  MoveL 585 to (127.63, -206.24, -1) mm, rotated rx -180 ry 0 rz 0 deg; joints [14.907, -52.311, 139.809, 14.927, -86.713, -0.372]
  MoveL 586 to (141.54, -192.34, -1) mm, rotated rx -180 ry 0 rz 0 deg; joints [15.844, -52.517, 140.53, 15.857, -87.219, -0.271]
  MoveL 587 to (229.23, -104.7, -1) mm, rotated rx -180 ry 0 rz 0 deg; joints [22.146, -53.586, 144.524, 22.139, -89.999, 0.626]
  MoveC 588 to (229.67, -104.52, -1) mm, rotated rx -180 ry 0 rz 0 deg; joints [22.166, -53.592, 144.549, 22.159, -90.017, 0.633] to (230.12, -104.7, -1) mm, rotated rx -180 ry 0 rz 0 deg; joints [22.165, -53.6, 144.584, 22.159, -90.042, 0.644]
  MoveL 589 to (230.57, -105.15, -1) mm, rotated rx 180 ry 0 rz 0 deg; joints [22.151, -53.609, 144.626, 22.144, -90.073, 0.656]
  MoveC 590 to (230.89, -105.47, -0.81) mm, rotated rx -180 ry 0 rz 0 deg; joints [22.141, -53.633, 144.659, 22.134, -90.081, 0.659] to (231.02, -105.6, -0.37) mm, rotated rx -180 ry 0 rz 0 deg; joints [22.136, -53.677, 144.678, 22.13, -90.057, 0.649]
  Set speed (500.0 mm/s)
  MoveL 591 to (231.02, -105.6, 5) mm, rotated rx 180 ry 0 rz 0 deg; joints [22.133, -54.178, 144.756, 22.127, -89.665, 0.49]
  MoveL 592 to (104.48, -103.86, 5) mm, rotated rx 180 ry 0 rz 0 deg; joints [19.74, -51.718, 135.968, 19.858, -83.72, -1.678]
  Set speed (25.4 mm/s)
  MoveL 593 to (104.48, -103.86, 1) mm, rotated rx 180 ry 0 rz 0 deg; joints [19.742, -51.399, 135.918, 19.85, -83.972, -1.587]
  MoveL 594 to (104.48, -103.86, -0.36) mm, rotated rx 180 ry 0 rz 0 deg; joints [19.743, -51.29, 135.9, 19.848, -84.058, -1.555]
  MoveC 595 to (104.61, -103.99, -0.81) mm, rotated rx -180 ry 0 rz 0 deg; joints [19.739, -51.258, 135.907, 19.842, -84.095, -1.542] to (104.93, -104.31, -1) mm, rotated rx -180 ry 0 rz 0 deg; joints [19.729, -51.252, 135.935, 19.831, -84.126, -1.529]
  Set speed (50.8 mm/s)
  MoveL 596 to (105.38, -104.76, -1) mm, rotated rx 180 ry 0 rz 0 deg; joints [19.715, -51.265, 135.978, 19.816, -84.154, -1.518]
  MoveC 597 to (105.57, -105.21, -1) mm, rotated rx -180 ry 0 rz 0 deg; joints [19.696, -51.273, 136.003, 19.797, -84.17, -1.51] to (105.38, -105.66, -1) mm, rotated rx 180 ry 0 rz 0 deg; joints [19.671, -51.272, 136.001, 19.771, -84.168, -1.509]
  MoveL 598 to (4.74, -206.24, -1) mm, rotated rx 180 ry 0 rz 0 deg; joints [13.359, -49.51, 130.795, 13.536, -80.653, -1.76]
  MoveL 599 to (106.34, -206.24, -1) mm, rotated rx -180 ry 0 rz 0 deg; joints [14.615, -51.88, 138.281, 14.652, -85.648, -0.638]
  MoveL 600 to (106.34, -104.7, -1) mm, rotated rx 180 ry 0 rz 0 deg; joints [19.735, -51.286, 136.045, 19.834, -84.198, -1.504]
  MoveL 601 to (105.38, -105.66, -1) mm, rotated rx -180 ry 0 rz 0 deg; joints [19.671, -51.272, 136.001, 19.771, -84.168, -1.509]
  MoveC 602 to (104.93, -105.85, -1) mm, rotated rx -180 ry 0 rz 0 deg; joints [19.654, -51.263, 135.974, 19.755, -84.15, -1.513] to (104.48, -105.66, -1) mm, rotated rx -180 ry 0 rz 0 deg; joints [19.655, -51.252, 135.937, 19.757, -84.126, -1.522]
  MoveL 603 to (104.03, -105.21, -1) mm, rotated rx -180 ry 0 rz 0 deg; joints [19.67, -51.239, 135.894, 19.772, -84.098, -1.534]
  MoveC 604 to (103.72, -104.89, -0.81) mm, rotated rx -180 ry 0 rz 0 deg; joints [19.68, -51.245, 135.866, 19.783, -84.067, -1.546] to (103.59, -104.76, -0.37) mm, rotated rx -180 ry 0 rz 0 deg; joints [19.683, -51.277, 135.859, 19.789, -84.031, -1.56]
  Set speed (500.0 mm/s)
  MoveL 605 to (103.59, -104.76, 5) mm, rotated rx -180 ry 0 rz 0 deg; joints [19.681, -51.705, 135.927, 19.799, -83.692, -1.682]
  MoveL 606 to (104.48, -231.14, 5) mm, rotated rx -180 ry 0 rz 0 deg; joints [13.293, -52.453, 138.67, 13.33, -85.449, -0.599]
  Set speed (25.4 mm/s)
  MoveL 607 to (104.48, -231.14, 1) mm, rotated rx -180 ry 0 rz 0 deg; joints [13.294, -52.119, 138.618, 13.326, -85.723, -0.534]
  MoveL 608 to (104.48, -231.14, -0.37) mm, rotated rx -180 ry 0 rz 0 deg; joints [13.295, -52.005, 138.599, 13.325, -85.816, -0.512]
  MoveC 609 to (104.61, -231.27, -0.81) mm, rotated rx -180 ry 0 rz 0 deg; joints [13.29, -51.971, 138.605, 13.32, -85.855, -0.503] to (104.93, -231.59, -1) mm, rotated rx -180 ry 0 rz 0 deg; joints [13.277, -51.963, 138.631, 13.306, -85.888, -0.494]
  Set speed (50.8 mm/s)
  MoveL 610 to (105.38, -232.04, -1) mm, rotated rx 180 ry 0 rz 0 deg; joints [13.259, -51.974, 138.671, 13.288, -85.916, -0.487]
  MoveC 611 to (105.57, -232.49, -1) mm, rotated rx -180 ry 0 rz 0 deg; joints [13.238, -51.98, 138.692, 13.266, -85.93, -0.482] to (105.38, -232.94, -1) mm, rotated rx -180 ry 0 rz 0 deg; joints [13.212, -51.978, 138.686, 13.241, -85.926, -0.481]
  MoveL 612 to (4.74, -333.52, -1) mm, rotated rx -180 ry 0 rz 0 deg; joints [7.16, -50.024, 132.531, 7.231, -81.696, -0.668]
  MoveL 613 to (106.34, -333.52, -1) mm, rotated rx 180 ry 0 rz 0 deg; joints [7.853, -52.311, 140.109, 7.859, -86.949, -0.029]
  MoveL 614 to (106.34, -231.98, -1) mm, rotated rx 180 ry 0 rz 0 deg; joints [13.274, -51.994, 138.739, 13.302, -85.963, -0.476]
  MoveL 615 to (105.38, -232.94, -1) mm, rotated rx -180 ry 0 rz 0 deg; joints [13.212, -51.978, 138.686, 13.241, -85.926, -0.481]
  MoveC 616 to (104.93, -233.12, -1) mm, rotated rx 180 ry 0 rz 0 deg; joints [13.197, -51.969, 138.657, 13.226, -85.905, -0.485] to (104.48, -232.94, -1) mm, rotated rx -180 ry 0 rz 0 deg; joints [13.201, -51.959, 138.621, 13.23, -85.881, -0.491]
  MoveL 617 to (104.03, -232.49, -1) mm, rotated rx 180 ry 0 rz 0 deg; joints [13.219, -51.948, 138.581, 13.249, -85.853, -0.499]
  MoveC 618 to (103.72, -232.17, -0.81) mm, rotated rx -180 ry 0 rz 0 deg; joints [13.232, -51.956, 138.555, 13.262, -85.82, -0.507] to (103.59, -232.04, -0.37) mm, rotated rx -180 ry 0 rz 0 deg; joints [13.237, -51.99, 138.549, 13.268, -85.781, -0.517]
  Set speed (500.0 mm/s)
  MoveL 619 to (103.59, -232.04, 5) mm, rotated rx 180 ry 0 rz 0 deg; joints [13.235, -52.438, 138.62, 13.272, -85.415, -0.604]
  MoveL 620 to (125.72, -232.7, 5) mm, rotated rx 180 ry 0 rz 0 deg; joints [13.477, -52.9, 140.23, 13.496, -86.534, -0.351]
  Set speed (25.4 mm/s)
  MoveL 621 to (125.72, -232.7, 1) mm, rotated rx 180 ry 0 rz 0 deg; joints [13.479, -52.557, 140.176, 13.494, -86.816, -0.283]
  MoveL 622 to (125.72, -232.7, -0.36) mm, rotated rx -180 ry 0 rz 0 deg; joints [13.479, -52.44, 140.158, 13.494, -86.911, -0.26]
  MoveC 623 to (125.91, -232.7, -0.81) mm, rotated rx 180 ry 0 rz 0 deg; joints [13.482, -52.405, 140.165, 13.496, -86.952, -0.25] to (126.35, -232.7, -1) mm, rotated rx -180 ry 0 rz 0 deg; joints [13.488, -52.398, 140.195, 13.501, -86.988, -0.242]
  Set speed (50.8 mm/s)
  MoveL 624 to (126.99, -232.7, -1) mm, rotated rx -180 ry 0 rz 0 deg; joints [13.496, -52.41, 140.24, 13.509, -87.021, -0.234]
  MoveC 625 to (127.44, -232.89, -1) mm, rotated rx 180 ry 0 rz 0 deg; joints [13.492, -52.419, 140.276, 13.504, -87.046, -0.228] to (127.62, -233.33, -1) mm, rotated rx -180 ry 0 rz 0 deg; joints [13.47, -52.425, 140.297, 13.482, -87.061, -0.224]
  MoveL 626 to (127.62, -333.52, -1) mm, rotated rx -180 ry 0 rz 0 deg; joints [8.016, -52.719, 141.661, 8.015, -88.082, 0.125]
  MoveL 627 to (229.22, -231.98, -1) mm, rotated rx -180 ry 0 rz 0 deg; joints [14.984, -54.068, 147.425, 14.991, -92.374, 1.14]
  MoveL 628 to (127.63, -231.98, -1) mm, rotated rx 180 ry 0 rz 0 deg; joints [13.542, -52.419, 140.273, 13.555, -87.044, -0.231]
  MoveL 629 to (127.62, -233.33, -1) mm, rotated rx -180 ry 0 rz 0 deg; joints [13.47, -52.425, 140.297, 13.482, -87.061, -0.224]
  MoveC 630 to (127.44, -233.78, -1) mm, rotated rx 180 ry 0 rz 0 deg; joints [13.444, -52.423, 140.291, 13.456, -87.057, -0.224] to (126.99, -233.97, -1) mm, rotated rx 180 ry 0 rz 0 deg; joints [13.428, -52.415, 140.262, 13.441, -87.036, -0.228]
  MoveL 631 to (126.35, -233.97, -1) mm, rotated rx -180 ry 0 rz 0 deg; joints [13.42, -52.403, 140.216, 13.433, -87.004, -0.236]
  MoveC 632 to (125.91, -233.97, -0.81) mm, rotated rx 180 ry 0 rz 0 deg; joints [13.414, -52.41, 140.187, 13.428, -86.968, -0.244] to (125.72, -233.97, -0.37) mm, rotated rx 180 ry 0 rz 0 deg; joints [13.412, -52.445, 140.179, 13.426, -86.927, -0.254]
  Set speed (500.0 mm/s)
  MoveL 633 to (125.72, -233.97, 5) mm, rotated rx -180 ry 0 rz 0 deg; joints [13.409, -52.905, 140.252, 13.428, -86.549, -0.344]
  MoveL 634 to (79.16, -230.07, 5) mm, rotated rx -180 ry 0 rz 0 deg; joints [13.042, -51.892, 136.807, 13.105, -84.177, -0.879]
  Set speed (25.4 mm/s)
  MoveL 635 to (79.16, -230.08, 1) mm, rotated rx 180 ry 0 rz 0 deg; joints [13.043, -51.568, 136.756, 13.1, -84.443, -0.817]
  MoveL 636 to (79.16, -230.08, -0.36) mm, rotated rx 180 ry 0 rz 0 deg; joints [13.044, -51.458, 136.738, 13.099, -84.533, -0.796]
  MoveC 637 to (79.16, -230.26, -0.81) mm, rotated rx 180 ry 0 rz 0 deg; joints [13.035, -51.422, 136.735, 13.089, -84.565, -0.788] to (79.16, -230.71, -1) mm, rotated rx 180 ry 0 rz 0 deg; joints [13.012, -51.409, 136.74, 13.065, -84.582, -0.782]
  Set speed (50.8 mm/s)
  MoveL 638 to (79.16, -231.34, -1) mm, rotated rx -180 ry 0 rz 0 deg; joints [12.979, -51.412, 136.751, 13.033, -84.589, -0.778]
  MoveC 639 to (78.98, -231.79, -1) mm, rotated rx 180 ry 0 rz 0 deg; joints [12.954, -51.41, 136.745, 13.007, -84.585, -0.777] to (78.53, -231.98, -1) mm, rotated rx -180 ry 0 rz 0 deg; joints [12.939, -51.401, 136.715, 12.993, -84.564, -0.78]
  MoveL 640 to (-23.07, -231.98, -1) mm, rotated rx -180 ry 0 rz 0 deg; joints [11.845, -48.917, 129.119, 12.043, -79.543, -1.763]
  MoveL 641 to (-23.07, -333.52, -1) mm, rotated rx -180 ry 0 rz 0 deg; joints [6.991, -49.311, 130.403, 7.088, -80.29, -0.823]
  MoveL 642 to (-9.16, -319.62, -1) mm, rotated rx 180 ry 0 rz 0 deg; joints [7.755, -49.632, 131.334, 7.849, -80.908, -0.857]
  MoveL 643 to (78.53, -231.98, -1) mm, rotated rx -180 ry 0 rz 0 deg; joints [12.939, -51.401, 136.715, 12.993, -84.564, -0.78]
  MoveC 644 to (78.98, -231.79, -1) mm, rotated rx 180 ry 0 rz 0 deg; joints [12.954, -51.41, 136.745, 13.007, -84.585, -0.777] to (79.43, -231.98, -1) mm, rotated rx -180 ry 0 rz 0 deg; joints [12.95, -51.42, 136.781, 13.003, -84.609, -0.771]
  MoveL 645 to (79.88, -232.43, -1) mm, rotated rx -180 ry 0 rz 0 deg; joints [12.932, -51.432, 136.821, 12.984, -84.637, -0.763]
  MoveC 646 to (80.19, -232.75, -0.81) mm, rotated rx 180 ry 0 rz 0 deg; joints [12.92, -51.456, 136.852, 12.971, -84.644, -0.76] to (80.32, -232.88, -0.37) mm, rotated rx 180 ry 0 rz 0 deg; joints [12.914, -51.496, 136.87, 12.967, -84.622, -0.765]
  Set speed (500.0 mm/s)
  MoveL 647 to (80.32, -232.88, 5) mm, rotated rx -180 ry 0 rz 0 deg; joints [12.912, -51.931, 136.939, 12.972, -84.265, -0.847]
  MoveL 648 to (-41.36, -230.18, 5) mm, rotated rx -180 ry 0 rz 0 deg; joints [11.749, -48.837, 127.757, 11.997, -78.285, -2.017]
  Set speed (25.4 mm/s)
  MoveL 649 to (-41.36, -230.18, 1) mm, rotated rx 180 ry 0 rz 0 deg; joints [11.75, -48.554, 127.71, 11.988, -78.517, -1.967]
  MoveL 650 to (-41.36, -230.18, -0.37) mm, rotated rx -180 ry 0 rz 0 deg; joints [11.751, -48.458, 127.694, 11.985, -78.595, -1.951]
  MoveC 651 to (-41.23, -230.32, -0.81) mm, rotated rx -180 ry 0 rz 0 deg; joints [11.746, -48.43, 127.701, 11.979, -78.629, -1.942] to (-40.91, -230.63, -1) mm, rotated rx 180 ry 0 rz 0 deg; joints [11.734, -48.428, 127.728, 11.966, -78.658, -1.934]
  Set speed (50.8 mm/s)
  MoveL 652 to (-40.46, -231.08, -1) mm, rotated rx -180 ry 0 rz 0 deg; joints [11.718, -48.442, 127.77, 11.948, -78.684, -1.925]
  MoveC 653 to (-40.27, -231.53, -1) mm, rotated rx -180 ry 0 rz 0 deg; joints [11.699, -48.45, 127.791, 11.928, -78.697, -1.919] to (-40.46, -231.98, -1) mm, rotated rx 180 ry 0 rz 0 deg; joints [11.676, -48.447, 127.784, 11.905, -78.691, -1.915]
  MoveL 654 to (-142.06, -333.52, -1) mm, rotated rx -180 ry 0 rz 0 deg; joints [6.349, -45.884, 120.993, 6.59, -74.333, -1.418]
  MoveL 655 to (-40.46, -333.52, -1) mm, rotated rx -180 ry 0 rz 0 deg; joints [6.889, -48.847, 129.06, 7.004, -79.415, -0.916]
  MoveL 656 to (-40.46, -231.98, -1) mm, rotated rx 180 ry 0 rz 0 deg; joints [11.676, -48.447, 127.784, 11.905, -78.691, -1.915]
  MoveC 657 to (-40.27, -231.53, -1) mm, rotated rx 180 ry 0 rz 0 deg; joints [11.699, -48.45, 127.791, 11.928, -78.697, -1.919] to (-39.82, -231.35, -1) mm, rotated rx -180 ry 0 rz 0 deg; joints [11.712, -48.461, 127.823, 11.94, -78.717, -1.917]
  MoveL 658 to (-39.19, -231.34, -1) mm, rotated rx 180 ry 0 rz 0 deg; joints [11.718, -48.478, 127.872, 11.945, -78.748, -1.911]
  MoveC 659 to (-38.74, -231.35, -0.81) mm, rotated rx -180 ry 0 rz 0 deg; joints [11.722, -48.504, 127.909, 11.949, -78.759, -1.91] to (-38.55, -231.34, -0.37) mm, rotated rx -180 ry 0 rz 0 deg; joints [11.724, -48.541, 127.928, 11.951, -78.742, -1.914]
  Set speed (500.0 mm/s)
  MoveL 660 to (-38.55, -231.34, 5) mm, rotated rx -180 ry 0 rz 0 deg; joints [11.722, -48.921, 127.991, 11.963, -78.431, -1.98]
  MoveL 661 to (-67.63, -230.07, 5) mm, rotated rx -180 ry 0 rz 0 deg; joints [11.505, -48.089, 125.716, 11.806, -77.01, -2.241]
  Set speed (25.4 mm/s)
  MoveL 662 to (-67.63, -230.07, 1) mm, rotated rx -180 ry 0 rz 0 deg; joints [11.507, -47.814, 125.67, 11.797, -77.235, -2.193]
  MoveL 663 to (-67.63, -230.07, -0.36) mm, rotated rx -180 ry 0 rz 0 deg; joints [11.507, -47.72, 125.654, 11.794, -77.312, -2.177]
  MoveC 664 to (-67.63, -230.26, -0.81) mm, rotated rx -180 ry 0 rz 0 deg; joints [11.499, -47.69, 125.652, 11.784, -77.338, -2.169] to (-67.63, -230.71, -1) mm, rotated rx -180 ry 0 rz 0 deg; joints [11.479, -47.679, 125.657, 11.763, -77.352, -2.162]
  Set speed (50.8 mm/s)
  MoveL 665 to (-67.63, -231.34, -1) mm, rotated rx -180 ry 0 rz 0 deg; joints [11.45, -47.683, 125.667, 11.733, -77.358, -2.154]
  MoveC 666 to (-67.82, -231.79, -1) mm, rotated rx -180 ry 0 rz 0 deg; joints [11.428, -47.68, 125.659, 11.71, -77.352, -2.151] to (-68.27, -231.98, -1) mm, rotated rx 180 ry 0 rz 0 deg; joints [11.415, -47.668, 125.627, 11.698, -77.332, -2.152]
  MoveL 667 to (-169.87, -231.98, -1) mm, rotated rx -180 ry 0 rz 0 deg; joints [10.552, -44.559, 117.485, 11.074, -72.355, -2.961]
  MoveL 668 to (-169.87, -333.52, -1) mm, rotated rx 180 ry 0 rz 0 deg; joints [6.216, -45.001, 118.713, 6.498, -72.941, -1.547]
  MoveL 669 to (-68.27, -231.98, -1) mm, rotated rx -180 ry 0 rz 0 deg; joints [11.415, -47.668, 125.627, 11.698, -77.332, -2.152]
  MoveC 670 to (-67.82, -231.79, -1) mm, rotated rx 180 ry 0 rz 0 deg; joints [11.428, -47.68, 125.659, 11.71, -77.352, -2.151] to (-67.37, -231.98, -1) mm, rotated rx 180 ry 0 rz 0 deg; joints [11.423, -47.694, 125.697, 11.705, -77.376, -2.145]
  MoveL 671 to (-66.92, -232.43, -1) mm, rotated rx -180 ry 0 rz 0 deg; joints [11.407, -47.709, 125.739, 11.687, -77.402, -2.136]
  MoveC 672 to (-66.61, -232.75, -0.81) mm, rotated rx -180 ry 0 rz 0 deg; joints [11.395, -47.732, 125.771, 11.675, -77.409, -2.131] to (-66.47, -232.88, -0.37) mm, rotated rx 180 ry 0 rz 0 deg; joints [11.39, -47.768, 125.789, 11.67, -77.392, -2.134]
  Set speed (500.0 mm/s)
  MoveL 673 to (-66.47, -232.88, 5) mm, rotated rx -180 ry 0 rz 0 deg; joints [11.389, -48.137, 125.85, 11.682, -77.09, -2.198]
  MoveL 674 to (-186.46, -230.18, 5) mm, rotated rx 180 ry 0 rz 0 deg; joints [10.497, -44.371, 116.15, 11.088, -71.226, -3.176]
  Set speed (25.4 mm/s)
  MoveL 675 to (-186.46, -230.18, 1) mm, rotated rx 180 ry 0 rz 0 deg; joints [10.498, -44.126, 116.107, 11.076, -71.425, -3.135]
  MoveL 676 to (-186.46, -230.18, -0.36) mm, rotated rx -180 ry 0 rz 0 deg; joints [10.498, -44.042, 116.092, 11.072, -71.493, -3.121]
  MoveC 677 to (-186.33, -230.32, -0.81) mm, rotated rx -180 ry 0 rz 0 deg; joints [10.494, -44.019, 116.1, 11.066, -71.522, -3.114] to (-186.01, -230.63, -1) mm, rotated rx 180 ry 0 rz 0 deg; joints [10.483, -44.02, 116.129, 11.053, -71.549, -3.104]
  Set speed (50.8 mm/s)
  MoveL 678 to (-185.56, -231.08, -1) mm, rotated rx 180 ry 0 rz 0 deg; joints [10.468, -44.038, 116.174, 11.035, -71.575, -3.094]
  MoveC 679 to (-185.38, -231.53, -1) mm, rotated rx -180 ry 0 rz 0 deg; joints [10.451, -44.047, 116.196, 11.016, -71.587, -3.086] to (-185.56, -231.98, -1) mm, rotated rx 180 ry 0 rz 0 deg; joints [10.431, -44.043, 116.187, 10.995, -71.581, -3.081]
  MoveL 680 to (-287.16, -333.52, -1) mm, rotated rx -180 ry 0 rz 0 deg; joints [5.71, -40.933, 108.684, 6.2, -66.998, -2.071]
  MoveL 681 to (-185.56, -333.52, -1) mm, rotated rx -180 ry 0 rz 0 deg; joints [6.143, -44.489, 117.411, 6.45, -72.154, -1.618]
  MoveL 682 to (-185.56, -231.98, -1) mm, rotated rx -180 ry 0 rz 0 deg; joints [10.431, -44.043, 116.187, 10.995, -71.581, -3.081]
  MoveC 683 to (-185.38, -231.53, -1) mm, rotated rx 180 ry 0 rz 0 deg; joints [10.451, -44.046, 116.196, 11.016, -71.587, -3.086] to (-184.93, -231.34, -1) mm, rotated rx -180 ry 0 rz 0 deg; joints [10.462, -44.06, 116.23, 11.026, -71.608, -3.085]
  MoveL 684 to (-184.29, -231.34, -1) mm, rotated rx -180 ry 0 rz 0 deg; joints [10.467, -44.081, 116.283, 11.03, -71.639, -3.081]
  MoveC 685 to (-183.84, -231.35, -0.81) mm, rotated rx 180 ry 0 rz 0 deg; joints [10.47, -44.108, 116.322, 11.032, -71.652, -3.079] to (-183.66, -231.35, -0.37) mm, rotated rx 180 ry 0 rz 0 deg; joints [10.472, -44.142, 116.343, 11.035, -71.639, -3.082]
  Set speed (500.0 mm/s)
  MoveL 686 to (-183.66, -231.35, 5) mm, rotated rx 180 ry 0 rz 0 deg; joints [10.47, -44.472, 116.401, 11.05, -71.371, -3.137]
  MoveL 687 to (-212.74, -230.07, 5) mm, rotated rx -180 ry 0 rz 0 deg; joints [10.302, -43.475, 113.946, 10.971, -69.93, -3.375]
  Set speed (25.4 mm/s)
  MoveL 688 to (-212.74, -230.07, 1) mm, rotated rx -180 ry 0 rz 0 deg; joints [10.303, -43.235, 113.903, 10.958, -70.124, -3.336]
  MoveL 689 to (-212.74, -230.08, -0.36) mm, rotated rx 180 ry 0 rz 0 deg; joints [10.304, -43.153, 113.889, 10.954, -70.19, -3.322]
  MoveC 690 to (-212.74, -230.26, -0.81) mm, rotated rx 180 ry 0 rz 0 deg; joints [10.296, -43.127, 113.887, 10.944, -70.213, -3.315] to (-212.74, -230.71, -1) mm, rotated rx 180 ry 0 rz 0 deg; joints [10.278, -43.118, 113.891, 10.924, -70.225, -3.306]
  Set speed (50.8 mm/s)
  MoveL 691 to (-212.74, -231.35, -1) mm, rotated rx 180 ry 0 rz 0 deg; joints [10.252, -43.122, 113.901, 10.896, -70.23, -3.296]
  MoveC 692 to (-212.92, -231.79, -1) mm, rotated rx 180 ry 0 rz 0 deg; joints [10.232, -43.118, 113.892, 10.876, -70.223, -3.29] to (-213.37, -231.98, -1) mm, rotated rx -180 ry 0 rz 0 deg; joints [10.221, -43.104, 113.857, 10.865, -70.202, -3.291]
  MoveL 693 to (-314.97, -231.98, -1) mm, rotated rx -180 ry 0 rz 0 deg; joints [9.523, -39.404, 104.979, 10.506, -65.066, -4.052]
  MoveL 694 to (-314.97, -333.52, -1) mm, rotated rx -180 ry 0 rz 0 deg; joints [5.602, -39.884, 106.192, 6.15, -65.559, -2.195]
  MoveL 695 to (-213.37, -231.98, -1) mm, rotated rx -180 ry 0 rz 0 deg; joints [10.221, -43.104, 113.857, 10.865, -70.202, -3.291]
  MoveC 696 to (-212.92, -231.79, -1) mm, rotated rx -180 ry 0 rz 0 deg; joints [10.232, -43.118, 113.892, 10.876, -70.223, -3.29] to (-212.47, -231.98, -1) mm, rotated rx -180 ry 0 rz 0 deg; joints [10.228, -43.135, 113.933, 10.869, -70.247, -3.284]
  MoveL 697 to (-212.03, -232.43, -1) mm, rotated rx 180 ry 0 rz 0 deg; joints [10.213, -43.153, 113.978, 10.852, -70.272, -3.273]
  MoveC 698 to (-211.71, -232.75, -0.81) mm, rotated rx -180 ry 0 rz 0 deg; joints [10.202, -43.176, 114.011, 10.839, -70.281, -3.268] to (-211.58, -232.88, -0.37) mm, rotated rx 180 ry 0 rz 0 deg; joints [10.198, -43.209, 114.029, 10.836, -70.267, -3.269]
  Set speed (500.0 mm/s)
  MoveL 699 to (-211.58, -232.88, 5) mm, rotated rx 180 ry 0 rz 0 deg; joints [10.196, -43.531, 114.086, 10.852, -70.006, -3.321]
  MoveL 700 to (-331.86, -230.18, 5) mm, rotated rx -180 ry 0 rz 0 deg; joints [9.482, -39.061, 103.475, 10.563, -63.921, -4.269]
  Set speed (25.4 mm/s)
  MoveL 701 to (-331.86, -230.18, 1) mm, rotated rx -180 ry 0 rz 0 deg; joints [9.483, -38.844, 103.433, 10.548, -64.094, -4.233]
  MoveL 702 to (-331.86, -230.18, -0.37) mm, rotated rx -180 ry 0 rz 0 deg; joints [9.483, -38.769, 103.419, 10.543, -64.153, -4.221]
  MoveC 703 to (-331.73, -230.32, -0.81) mm, rotated rx -180 ry 0 rz 0 deg; joints [9.479, -38.751, 103.428, 10.536, -64.18, -4.214] to (-331.41, -230.63, -1) mm, rotated rx -180 ry 0 rz 0 deg; joints [9.469, -38.755, 103.46, 10.523, -64.207, -4.204]
  Set speed (50.8 mm/s)
  MoveL 704 to (-330.96, -231.08, -1) mm, rotated rx -180 ry 0 rz 0 deg; joints [9.455, -38.775, 103.508, 10.505, -64.233, -4.191]
  MoveC 705 to (-330.77, -231.53, -1) mm, rotated rx 180 ry 0 rz 0 deg; joints [9.439, -38.785, 103.532, 10.486, -64.245, -4.181] to (-330.96, -231.98, -1) mm, rotated rx -180 ry 0 rz 0 deg; joints [9.421, -38.781, 103.522, 10.466, -64.238, -4.174]
  MoveL 706 to (-432.56, -333.52, -1) mm, rotated rx -180 ry 0 rz 0 deg; joints [5.186, -35.051, 95.037, 6.032, -59.253, -2.741]
  MoveL 707 to (-330.96, -333.52, -1) mm, rotated rx -180 ry 0 rz 0 deg; joints [5.542, -39.266, 104.737, 6.125, -64.724, -2.267]
  MoveL 708 to (-330.96, -231.98, -1) mm, rotated rx 180 ry 0 rz 0 deg; joints [9.421, -38.781, 103.522, 10.466, -64.238, -4.174]
  MoveC 709 to (-330.78, -231.53, -1) mm, rotated rx -180 ry 0 rz 0 deg; joints [9.439, -38.785, 103.532, 10.486, -64.245, -4.181] to (-330.33, -231.35, -1) mm, rotated rx -180 ry 0 rz 0 deg; joints [9.449, -38.802, 103.57, 10.495, -64.267, -4.181]
  MoveL 710 to (-329.69, -231.35, -1) mm, rotated rx 180 ry 0 rz 0 deg; joints [9.453, -38.827, 103.629, 10.497, -64.3, -4.177]
  MoveC 711 to (-329.24, -231.34, -0.81) mm, rotated rx -180 ry 0 rz 0 deg; joints [9.456, -38.855, 103.672, 10.498, -64.315, -4.175] to (-329.06, -231.35, -0.37) mm, rotated rx 180 ry 0 rz 0 deg; joints [9.457, -38.887, 103.694, 10.5, -64.306, -4.177]
  Set speed (500.0 mm/s)
  MoveL 712 to (-329.06, -231.35, 5) mm, rotated rx 180 ry 0 rz 0 deg; joints [9.456, -39.179, 103.749, 10.52, -64.072, -4.225]
  MoveL 713 to (-359.49, -230.07, 5) mm, rotated rx -180 ry 0 rz 0 deg; joints [9.315, -37.948, 100.91, 10.51, -62.48, -4.485]
  Set speed (25.4 mm/s)
  MoveL 714 to (-359.49, -230.08, 1) mm, rotated rx 180 ry 0 rz 0 deg; joints [9.316, -37.735, 100.869, 10.495, -62.649, -4.45]
  MoveL 715 to (-359.49, -230.07, -0.37) mm, rotated rx 180 ry 0 rz 0 deg; joints [9.316, -37.662, 100.854, 10.49, -62.706, -4.438]
  MoveC 716 to (-359.49, -230.26, -0.81) mm, rotated rx 180 ry 0 rz 0 deg; joints [9.309, -37.639, 100.852, 10.48, -62.726, -4.43] to (-359.49, -230.71, -1) mm, rotated rx -180 ry 0 rz 0 deg; joints [9.293, -37.632, 100.857, 10.461, -62.737, -4.42]
  Set speed (50.8 mm/s)
  MoveL 717 to (-359.49, -231.34, -1) mm, rotated rx 180 ry 0 rz 0 deg; joints [9.269, -37.636, 100.867, 10.434, -62.741, -4.407]
  MoveC 718 to (-359.68, -231.79, -1) mm, rotated rx -180 ry 0 rz 0 deg; joints [9.251, -37.631, 100.856, 10.414, -62.733, -4.399] to (-360.13, -231.98, -1) mm, rotated rx -180 ry 0 rz 0 deg; joints [9.242, -37.614, 100.817, 10.405, -62.711, -4.399]
  MoveL 719 to (-432.56, -231.98, -1) mm, rotated rx -180 ry 0 rz 0 deg; joints [8.824, -34.532, 93.796, 10.325, -58.8, -4.984]
  MoveL 720 to (-460.37, -231.98, -1) mm, rotated rx -180 ry 0 rz 0 deg; joints [8.673, -33.271, 90.967, 10.324, -57.244, -5.224]
  MoveL 721 to (-460.37, -333.52, -1) mm, rotated rx -180 ry 0 rz 0 deg; joints [5.097, -33.801, 92.222, 6.028, -57.692, -2.881]
  MoveL 722 to (-358.77, -231.98, -1) mm, rotated rx -180 ry 0 rz 0 deg; joints [9.25, -37.669, 100.944, 10.408, -62.782, -4.388]
  MoveL 723 to (-360.13, -231.98, -1) mm, rotated rx -180 ry 0 rz 0 deg; joints [9.242, -37.614, 100.817, 10.405, -62.711, -4.399]
  MoveC 724 to (-360.58, -231.79, -1) mm, rotated rx 180 ry 0 rz 0 deg; joints [9.246, -37.595, 100.772, 10.413, -62.686, -4.406] to (-360.76, -231.35, -1) mm, rotated rx -180 ry 0 rz 0 deg; joints [9.261, -37.584, 100.748, 10.431, -62.673, -4.417]
  MoveL 725 to (-360.76, -230.71, -1) mm, rotated rx -180 ry 0 rz 0 deg; joints [9.285, -37.58, 100.738, 10.458, -62.67, -4.43]
  MoveC 726 to (-360.76, -230.26, -0.81) mm, rotated rx 180 ry 0 rz 0 deg; joints [9.302, -37.588, 100.733, 10.478, -62.659, -4.44] to (-360.76, -230.08, -0.37) mm, rotated rx -180 ry 0 rz 0 deg; joints [9.308, -37.61, 100.735, 10.488, -62.639, -4.448]
  Set speed (500.0 mm/s)
  MoveL 727 to (-360.76, -230.07, 5) mm, rotated rx -180 ry 0 rz 0 deg; joints [9.307, -37.896, 100.79, 10.508, -62.413, -4.495]
  MoveL 728 to (253.69, -232.63, 5) mm, rotated rx -180 ry 0 rz 0 deg; joints [15.334, -54.969, 149.213, 15.353, -93.223, 1.395]
  Set speed (25.4 mm/s)
  MoveL 729 to (253.69, -232.63, 1) mm, rotated rx -180 ry 0 rz 0 deg; joints [15.336, -54.56, 149.15, 15.361, -93.558, 1.487]
  MoveL 730 to (253.69, -232.63, -0.36) mm, rotated rx 180 ry 0 rz 0 deg; joints [15.337, -54.42, 149.129, 15.363, -93.671, 1.519]
  MoveC 731 to (253.82, -232.77, -0.81) mm, rotated rx -180 ry 0 rz 0 deg; joints [15.332, -54.376, 149.133, 15.359, -93.718, 1.531] to (254.14, -233.08, -1) mm, rotated rx -180 ry 0 rz 0 deg; joints [15.318, -54.361, 149.157, 15.346, -93.757, 1.541]
  Set speed (50.8 mm/s)
  MoveL 732 to (254.59, -233.53, -1) mm, rotated rx -180 ry 0 rz 0 deg; joints [15.298, -54.366, 149.196, 15.327, -93.789, 1.548]
  MoveC 733 to (254.77, -233.98, -1) mm, rotated rx -180 ry 0 rz 0 deg; joints [15.274, -54.369, 149.217, 15.303, -93.808, 1.551] to (254.58, -234.43, -1) mm, rotated rx -180 ry 0 rz 0 deg; joints [15.244, -54.368, 149.213, 15.273, -93.805, 1.547]
  MoveL 734 to (155.44, -333.52, -1) mm, rotated rx -180 ry 0 rz 0 deg; joints [8.238, -53.209, 143.67, 8.233, -89.586, 0.338]
  MoveL 735 to (257.04, -333.52, -1) mm, rotated rx -180 ry 0 rz 0 deg; joints [9.168, -54.512, 150.851, 9.203, -95.388, 1.284]
  MoveL 736 to (257.04, -231.98, -1) mm, rotated rx -180 ry 0 rz 0 deg; joints [15.432, -54.389, 149.335, 15.463, -93.898, 1.59]
  MoveL 737 to (254.58, -234.43, -1) mm, rotated rx 180 ry 0 rz 0 deg; joints [15.244, -54.368, 149.213, 15.273, -93.805, 1.547]
  MoveC 738 to (254.14, -234.62, -1) mm, rotated rx -180 ry 0 rz 0 deg; joints [15.226, -54.364, 149.186, 15.254, -93.783, 1.54] to (253.69, -234.43, -1) mm, rotated rx -180 ry 0 rz 0 deg; joints [15.23, -54.358, 149.152, 15.257, -93.755, 1.532]
  MoveL 739 to (253.24, -233.98, -1) mm, rotated rx -180 ry 0 rz 0 deg; joints [15.249, -54.353, 149.113, 15.276, -93.723, 1.525]
  MoveC 740 to (252.92, -233.66, -0.81) mm, rotated rx -180 ry 0 rz 0 deg; joints [15.263, -54.368, 149.088, 15.289, -93.684, 1.516] to (252.79, -233.53, -0.37) mm, rotated rx -180 ry 0 rz 0 deg; joints [15.268, -54.412, 149.084, 15.294, -93.637, 1.503]
  Set speed (500.0 mm/s)
  MoveL 741 to (252.79, -233.53, 5) mm, rotated rx 180 ry 0 rz 0 deg; joints [15.266, -54.961, 149.168, 15.284, -93.189, 1.381]
  MoveL 742 to (272.52, -232.7, 5) mm, rotated rx -180 ry 0 rz 0 deg; joints [15.646, -55.172, 150.501, 15.684, -94.261, 1.711]
  Set speed (25.4 mm/s)
  MoveL 743 to (272.52, -232.7, 1) mm, rotated rx -180 ry 0 rz 0 deg; joints [15.648, -54.751, 150.436, 15.694, -94.605, 1.808]
  MoveL 744 to (272.52, -232.7, -0.37) mm, rotated rx -180 ry 0 rz 0 deg; joints [15.649, -54.607, 150.414, 15.697, -94.722, 1.841]
  MoveC 745 to (272.7, -232.7, -0.81) mm, rotated rx -180 ry 0 rz 0 deg; joints [15.652, -54.561, 150.419, 15.702, -94.77, 1.855] to (273.15, -232.7, -1) mm, rotated rx 180 ry 0 rz 0 deg; joints [15.66, -54.546, 150.446, 15.711, -94.812, 1.868]
  Set speed (50.8 mm/s)
  MoveL 746 to (273.79, -232.7, -1) mm, rotated rx -180 ry 0 rz 0 deg; joints [15.671, -54.552, 150.489, 15.722, -94.847, 1.879]
  MoveC 747 to (274.24, -232.89, -1) mm, rotated rx -180 ry 0 rz 0 deg; joints [15.667, -54.556, 150.523, 15.719, -94.876, 1.887] to (274.42, -233.33, -1) mm, rotated rx -180 ry 0 rz 0 deg; joints [15.643, -54.558, 150.544, 15.696, -94.895, 1.889]
  MoveL 748 to (274.42, -333.52, -1) mm, rotated rx -180 ry 0 rz 0 deg; joints [9.348, -54.643, 152.055, 9.403, -96.444, 1.48]
  MoveL 749 to (376.02, -231.98, -1) mm, rotated rx 180 ry 0 rz 0 deg; joints [17.686, -54.899, 157.276, 18.017, -100.916, 4.074]
  MoveL 750 to (274.42, -231.98, -1) mm, rotated rx -180 ry 0 rz 0 deg; joints [15.726, -54.556, 150.519, 15.778, -94.87, 1.891]
  MoveL 751 to (274.42, -233.33, -1) mm, rotated rx -180 ry 0 rz 0 deg; joints [15.643, -54.558, 150.544, 15.696, -94.895, 1.889]
  MoveC 752 to (274.24, -233.78, -1) mm, rotated rx -180 ry 0 rz 0 deg; joints [15.612, -54.557, 150.54, 15.665, -94.893, 1.885] to (273.79, -233.97, -1) mm, rotated rx -180 ry 0 rz 0 deg; joints [15.593, -54.554, 150.513, 15.645, -94.871, 1.877]
  MoveL 753 to (273.15, -233.97, -1) mm, rotated rx 180 ry 0 rz 0 deg; joints [15.582, -54.548, 150.47, 15.633, -94.835, 1.866]
  MoveC 754 to (272.7, -233.97, -0.81) mm, rotated rx -180 ry 0 rz 0 deg; joints [15.574, -54.563, 150.443, 15.625, -94.794, 1.853] to (272.52, -233.97, -0.37) mm, rotated rx 180 ry 0 rz 0 deg; joints [15.571, -54.609, 150.438, 15.62, -94.745, 1.839]
  Set speed (500.0 mm/s)
  MoveL 755 to (272.52, -233.97, 5) mm, rotated rx -180 ry 0 rz 0 deg; joints [15.568, -55.175, 150.525, 15.607, -94.284, 1.71]
  MoveL 756 to (400.49, -232.63, 5) mm, rotated rx 180 ry 0 rz 30 deg; joints [27.528, -55.537, 151.799, 57.6, -92.472, 5.085]
  Set speed (25.4 mm/s)
  MoveL 757 to (400.49, -232.63, 1) mm, rotated rx 180 ry 0 rz 30 deg; joints [27.531, -55.103, 151.733, 57.617, -92.669, 5.397]
  MoveL 758 to (400.49, -232.63, -0.37) mm, rotated rx 180 ry 0 rz 30 deg; joints [27.532, -54.955, 151.71, 57.623, -92.736, 5.503]
  MoveC 759 to (400.62, -232.77, -0.81) mm, rotated rx -180 ry 0 rz 30 deg; joints [27.528, -54.907, 151.715, 57.622, -92.764, 5.547] to (400.93, -233.08, -1) mm, rotated rx -180 ry 0 rz 30 deg; joints [27.52, -54.89, 151.741, 57.615, -92.788, 5.583]
  Set speed (50.8 mm/s)
  MoveL 760 to (401.38, -233.53, -1) mm, rotated rx -180 ry 0 rz 30 deg; joints [27.508, -54.894, 151.784, 57.605, -92.81, 5.615]
  MoveC 761 to (401.57, -233.98, -1) mm, rotated rx -180 ry 0 rz 30 deg; joints [27.487, -54.897, 151.81, 57.585, -92.825, 5.634] to (401.38, -234.43, -1) mm, rotated rx -180 ry 0 rz 30 deg; joints [27.456, -54.896, 151.813, 57.554, -92.83, 5.634]
  MoveL 762 to (389.92, -245.89, -1) mm, rotated rx 180 ry 0 rz 30 deg; joints [26.46, -54.84, 151.457, 56.55, -92.765, 5.319]
  MoveL 763 to (302.23, -333.52, -1) mm, rotated rx -180 ry 0 rz 0 deg; joints [9.651, -54.783, 153.966, 9.746, -98.183, 1.821]
  MoveL 764 to (403.83, -333.52, -1) mm, rotated rx -180 ry 0 rz 30 deg; joints [21.529, -54.989, 154.813, 51.82, -95.213, 7.51]
  MoveL 765 to (403.83, -231.98, -1) mm, rotated rx -180 ry 0 rz 30 deg; joints [27.67, -54.908, 151.886, 57.77, -92.841, 5.701]
  MoveL 766 to (401.38, -234.43, -1) mm, rotated rx -180 ry 0 rz 30 deg; joints [27.456, -54.896, 151.813, 57.554, -92.83, 5.634]
  MoveC 767 to (400.93, -234.62, -1) mm, rotated rx -180 ry 0 rz 30 deg; joints [27.432, -54.894, 151.791, 57.529, -92.822, 5.617] to (400.48, -234.43, -1) mm, rotated rx -180 ry 0 rz 30 deg; joints [27.429, -54.89, 151.757, 57.526, -92.806, 5.591]
  MoveL 768 to (400.04, -233.98, -1) mm, rotated rx -180 ry 0 rz 30 deg; joints [27.442, -54.886, 151.714, 57.536, -92.784, 5.559]
  MoveC 769 to (399.72, -233.66, -0.81) mm, rotated rx -180 ry 0 rz 30 deg; joints [27.45, -54.903, 151.687, 57.543, -92.759, 5.523] to (399.59, -233.53, -0.37) mm, rotated rx -180 ry 0 rz 30 deg; joints [27.453, -54.95, 151.683, 57.544, -92.731, 5.479]
  Set speed (500.0 mm/s)
  MoveL 770 to (399.59, -233.53, 5) mm, rotated rx -180 ry 0 rz 30 deg; joints [27.45, -55.532, 151.771, 57.522, -92.467, 5.062]
  MoveL 771 to (441.13, 165.37, 5) mm, rotated rx 180 ry 0 rz 0 deg; joints [42.449, -55.095, 147.223, 42.443, -90.701, 1.708]
  Set speed (25.4 mm/s)
  MoveL 772 to (441.13, 165.37, 1) mm, rotated rx 180 ry 0 rz 0 deg; joints [42.453, -54.703, 147.163, 42.45, -90.946, 1.933]
  MoveL 773 to (441.13, 165.37, -0.36) mm, rotated rx -180 ry 0 rz 0 deg; joints [42.454, -54.569, 147.143, 42.452, -91.03, 2.009]
  MoveC 774 to (441.13, 165.55, -0.81) mm, rotated rx 180 ry 0 rz 0 deg; joints [42.463, -54.523, 147.127, 42.461, -91.051, 2.03] to (441.13, 166, -1) mm, rotated rx -180 ry 0 rz 0 deg; joints [42.483, -54.502, 147.102, 42.481, -91.049, 2.029]
  Set speed (50.8 mm/s)
  MoveL 775 to (441.13, 166.64, -1) mm, rotated rx 180 ry 0 rz 0 deg; joints [42.511, -54.496, 147.072, 42.509, -91.029, 2.013]
  MoveC 776 to (441.31, 167.09, -1) mm, rotated rx 180 ry 0 rz 0 deg; joints [42.538, -54.495, 147.06, 42.536, -91.021, 2.007] to (441.76, 167.27, -1) mm, rotated rx -180 ry 0 rz 0 deg; joints [42.565, -54.498, 147.075, 42.563, -91.028, 2.015]
  MoveL 777 to (467.16, 167.27, -1) mm, rotated rx -180 ry 0 rz 0 deg; joints [43.62, -54.76, 148.403, 43.635, -91.768, 2.785]
  MoveL 778 to (467.16, 205.37, -1) mm, rotated rx -180 ry 0 rz 0 deg; joints [45.267, -54.446, 146.502, 45.259, -90.578, 1.733]
  MoveL 779 to (390.96, 205.37, -1) mm, rotated rx -180 ry 0 rz 0 deg; joints [42.209, -53.48, 142.502, 42.219, -88.406, -0.385]
  MoveL 780 to (390.96, 192.67, -1) mm, rotated rx 180 ry 0 rz 0 deg; joints [41.674, -53.621, 143.12, 41.676, -88.756, -0.061]
  MoveL 781 to (340.16, 192.67, -1) mm, rotated rx 180 ry 0 rz 0 deg; joints [39.822, -52.856, 140.29, 39.871, -87.16, -1.373]
  MoveL 782 to (340.16, 205.37, -1) mm, rotated rx -180 ry 0 rz 0 deg; joints [40.352, -52.702, 139.687, 40.417, -86.834, -1.682]
  MoveL 783 to (263.96, 205.37, -1) mm, rotated rx -180 ry 0 rz 0 deg; joints [37.81, -51.342, 135.252, 38.02, -84.323, -3.475]
  MoveL 784 to (263.96, 192.67, -1) mm, rotated rx 180 ry 0 rz 0 deg; joints [37.29, -51.513, 135.834, 37.474, -84.616, -3.18]
  MoveL 785 to (213.16, 192.67, -1) mm, rotated rx 180 ry 0 rz 0 deg; joints [35.75, -50.494, 132.726, 36.066, -82.835, -4.292]
  MoveL 786 to (213.16, 205.37, -1) mm, rotated rx 180 ry 0 rz 0 deg; joints [36.262, -50.314, 132.155, 36.611, -82.562, -4.584]
  MoveL 787 to (136.96, 205.37, -1) mm, rotated rx 180 ry 0 rz 0 deg; joints [34.137, -48.596, 127.299, 34.754, -79.804, -6.14]
  MoveL 788 to (136.96, 192.67, -1) mm, rotated rx 180 ry 0 rz 0 deg; joints [33.638, -48.786, 127.855, 34.214, -80.052, -5.849]
  MoveL 789 to (86.16, 192.67, -1) mm, rotated rx 180 ry 0 rz 0 deg; joints [32.349, -47.533, 124.468, 33.137, -78.127, -6.827]
  MoveL 790 to (86.16, 205.37, -1) mm, rotated rx 180 ry 0 rz 0 deg; joints [32.838, -47.337, 123.92, 33.674, -77.895, -7.121]
  MoveL 791 to (9.96, 205.37, -1) mm, rotated rx 180 ry 0 rz 0 deg; joints [31.047, -45.28, 118.627, 32.276, -74.927, -8.531]
  MoveL 792 to (9.96, 167.27, -1) mm, rotated rx 180 ry 0 rz 0 deg; joints [29.612, -45.875, 120.213, 30.671, -75.564, -7.644]
  MoveL 793 to (35.36, 167.27, -1) mm, rotated rx -180 ry 0 rz 0 deg; joints [30.173, -46.576, 122.017, 31.103, -76.586, -7.19]
  MoveC 794 to (48.06, 179.97, -1) mm, rotated rx -180 ry 0 rz 0 deg; joints [30.952, -46.728, 122.384, 31.871, -76.871, -7.245] to (60.76, 167.27, -1) mm, rotated rx -180 ry 0 rz 0 deg; joints [30.754, -47.254, 123.791, 31.564, -77.595, -6.728]
  MoveL 795 to (162.36, 167.27, -1) mm, rotated rx -180 ry 0 rz 0 deg; joints [33.292, -49.737, 130.602, 33.702, -81.507, -4.783]
  MoveC 796 to (175.06, 179.97, -1) mm, rotated rx -180 ry 0 rz 0 deg; joints [34.154, -49.846, 130.876, 34.556, -81.72, -4.802] to (187.76, 167.27, -1) mm, rotated rx 180 ry 0 rz 0 deg; joints [33.986, -50.3, 132.235, 34.315, -82.453, -4.264]
  MoveL 797 to (289.36, 167.27, -1) mm, rotated rx -180 ry 0 rz 0 deg; joints [37.031, -52.302, 138.5, 37.123, -86.097, -2.022]
  MoveC 798 to (302.06, 179.97, -1) mm, rotated rx -180 ry 0 rz 0 deg; joints [37.987, -52.371, 138.677, 38.075, -86.22, -2.005] to (314.76, 167.27, -1) mm, rotated rx 180 ry 0 rz 0 deg; joints [37.867, -52.738, 139.999, 37.92, -86.968, -1.411]
  MoveL 799 to (416.36, 167.27, -1) mm, rotated rx 180 ry 0 rz 0 deg; joints [41.551, -54.205, 145.717, 41.541, -90.262, 1.275]
  MoveC 800 to (429.06, 179.97, -1) mm, rotated rx 180 ry 0 rz 0 deg; joints [42.61, -54.242, 145.787, 42.6, -90.267, 1.318] to (441.76, 167.27, -1) mm, rotated rx 180 ry 0 rz 0 deg; joints [42.565, -54.498, 147.075, 42.563, -91.028, 2.015]
  MoveC 801 to (441.58, 166.82, -1) mm, rotated rx 180 ry 0 rz 0 deg; joints [42.537, -54.5, 147.087, 42.536, -91.037, 2.021] to (441.13, 166.64, -1) mm, rotated rx 180 ry 0 rz 0 deg; joints [42.511, -54.496, 147.072, 42.509, -91.029, 2.013]
  MoveL 802 to (440.49, 166.64, -1) mm, rotated rx 180 ry 0 rz 0 deg; joints [42.485, -54.489, 147.038, 42.483, -91.01, 1.994]
  MoveC 803 to (440.04, 166.64, -0.81) mm, rotated rx -180 ry 0 rz 0 deg; joints [42.467, -54.503, 147.017, 42.464, -90.986, 1.97] to (439.86, 166.64, -0.37) mm, rotated rx -180 ry 0 rz 0 deg; joints [42.459, -54.544, 147.014, 42.456, -90.953, 1.939]
  Set speed (500.0 mm/s)
  MoveL 804 to (439.86, 166.64, 5) mm, rotated rx -180 ry 0 rz 0 deg; joints [42.454, -55.069, 147.094, 42.447, -90.625, 1.639]
  MoveL 805 to (441.13, 227.71, 5) mm, rotated rx 180 ry 0 rz 0 deg; joints [45.102, -54.463, 144.118, 45.102, -88.887, 0.028]
  Set speed (25.4 mm/s)
  MoveL 806 to (441.13, 227.71, 1) mm, rotated rx -180 ry 0 rz 0 deg; joints [45.105, -54.094, 144.062, 45.102, -89.107, 0.249]
  MoveL 807 to (441.13, 227.71, -0.37) mm, rotated rx -180 ry 0 rz 0 deg; joints [45.106, -53.969, 144.042, 45.101, -89.182, 0.324]
  MoveC 808 to (441.13, 227.9, -0.81) mm, rotated rx -180 ry 0 rz 0 deg; joints [45.114, -53.925, 144.026, 45.109, -89.202, 0.344] to (441.13, 228.34, -1) mm, rotated rx -180 ry 0 rz 0 deg; joints [45.133, -53.903, 144, 45.128, -89.199, 0.341]
  Set speed (50.8 mm/s)
  MoveL 809 to (441.13, 228.98, -1) mm, rotated rx -180 ry 0 rz 0 deg; joints [45.159, -53.896, 143.968, 45.154, -89.181, 0.323]
  MoveC 810 to (441.31, 229.43, -1) mm, rotated rx 180 ry 0 rz 0 deg; joints [45.184, -53.893, 143.954, 45.18, -89.173, 0.316] to (441.76, 229.62, -1) mm, rotated rx 180 ry 0 rz 0 deg; joints [45.21, -53.897, 143.968, 45.205, -89.18, 0.322]
  MoveL 811 to (467.16, 229.62, -1) mm, rotated rx -180 ry 0 rz 0 deg; joints [46.267, -54.209, 145.255, 46.256, -89.854, 1.028]
  MoveL 812 to (467.16, 267.72, -1) mm, rotated rx -180 ry 0 rz 0 deg; joints [47.769, -53.781, 143.239, 47.772, -88.767, -0.129]
  MoveL 813 to (390.96, 267.72, -1) mm, rotated rx -180 ry 0 rz 0 deg; joints [44.712, -52.699, 139.353, 44.792, -86.754, -2.084]
  MoveL 814 to (390.96, 255.01, -1) mm, rotated rx -180 ry 0 rz 0 deg; joints [44.219, -52.87, 140.01, 44.28, -87.082, -1.724]
  MoveL 815 to (340.16, 255.02, -1) mm, rotated rx 180 ry 0 rz 0 deg; joints [42.349, -52.042, 137.252, 42.494, -85.593, -2.962]
  MoveL 816 to (340.16, 267.72, -1) mm, rotated rx -180 ry 0 rz 0 deg; joints [42.841, -51.859, 136.608, 43.011, -85.285, -3.307]
  MoveL 817 to (263.96, 267.71, -1) mm, rotated rx 180 ry 0 rz 0 deg; joints [40.262, -50.427, 132.267, 40.626, -82.916, -5.031]
  MoveL 818 to (263.96, 255.01, -1) mm, rotated rx 180 ry 0 rz 0 deg; joints [39.776, -50.624, 132.891, 40.105, -83.198, -4.701]
  MoveL 819 to (213.16, 255.01, -1) mm, rotated rx -180 ry 0 rz 0 deg; joints [38.202, -49.564, 129.838, 38.694, -81.506, -5.791]
  MoveL 820 to (213.16, 267.72, -1) mm, rotated rx 180 ry 0 rz 0 deg; joints [38.682, -49.36, 129.225, 39.216, -81.24, -6.116]
  MoveL 821 to (136.96, 267.71, -1) mm, rotated rx 180 ry 0 rz 0 deg; joints [36.501, -47.594, 124.44, 37.35, -78.597, -7.665]
  MoveL 822 to (136.96, 255.01, -1) mm, rotated rx -180 ry 0 rz 0 deg; joints [36.031, -47.808, 125.04, 36.828, -78.842, -7.341]
  MoveL 823 to (86.16, 255.01, -1) mm, rotated rx 180 ry 0 rz 0 deg; joints [34.698, -46.527, 121.691, 35.742, -76.987, -8.331]
  MoveL 824 to (86.16, 267.71, -1) mm, rotated rx -180 ry 0 rz 0 deg; joints [35.161, -46.308, 121.098, 36.263, -76.755, -8.656]
  MoveL 825 to (9.96, 267.71, -1) mm, rotated rx -180 ry 0 rz 0 deg; joints [33.306, -44.215, 115.848, 34.853, -73.875, -10.103]
  MoveL 826 to (9.96, 229.61, -1) mm, rotated rx 180 ry 0 rz 0 deg; joints [31.939, -44.879, 117.573, 33.285, -74.519, -9.125]
  MoveL 827 to (35.36, 229.61, -1) mm, rotated rx 180 ry 0 rz 0 deg; joints [32.525, -45.592, 119.363, 33.725, -75.511, -8.655]
  MoveC 828 to (48.06, 242.31, -1) mm, rotated rx 180 ry 0 rz 0 deg; joints [33.292, -45.727, 119.677, 34.482, -75.778, -8.734] to (60.76, 229.61, -1) mm, rotated rx 180 ry 0 rz 0 deg; joints [33.131, -46.282, 121.121, 34.193, -76.488, -8.181]
  MoveL 829 to (162.36, 229.61, -1) mm, rotated rx -180 ry 0 rz 0 deg; joints [35.765, -48.822, 127.851, 36.363, -80.252, -6.207]
  MoveC 830 to (175.06, 242.31, -1) mm, rotated rx -180 ry 0 rz 0 deg; joints [36.607, -48.915, 128.07, 37.199, -80.449, -6.26] to (187.76, 229.61, -1) mm, rotated rx -180 ry 0 rz 0 deg; joints [36.481, -49.401, 129.46, 36.983, -81.156, -5.69]
  MoveL 831 to (289.36, 229.62, -1) mm, rotated rx -180 ry 0 rz 0 deg; joints [39.607, -51.489, 135.61, 39.808, -84.606, -3.488]
  MoveC 832 to (302.06, 242.32, -1) mm, rotated rx -180 ry 0 rz 0 deg; joints [40.533, -51.544, 135.73, 40.733, -84.716, -3.518] to (314.76, 229.61, -1) mm, rotated rx -180 ry 0 rz 0 deg; joints [40.459, -51.952, 137.076, 40.606, -85.424, -2.899]
  MoveL 833 to (416.36, 229.61, -1) mm, rotated rx 180 ry 0 rz 0 deg; joints [44.191, -53.559, 142.649, 44.2, -88.478, -0.362]
  MoveC 834 to (429.06, 242.31, -1) mm, rotated rx -180 ry 0 rz 0 deg; joints [45.207, -53.583, 142.66, 45.216, -88.48, -0.383] to (441.76, 229.61, -1) mm, rotated rx -180 ry 0 rz 0 deg; joints [45.21, -53.897, 143.968, 45.205, -89.18, 0.322]
  MoveC 835 to (441.58, 229.17, -1) mm, rotated rx 180 ry 0 rz 0 deg; joints [45.184, -53.9, 143.981, 45.179, -89.188, 0.33] to (441.13, 228.98, -1) mm, rotated rx 180 ry 0 rz 0 deg; joints [45.159, -53.896, 143.968, 45.154, -89.181, 0.323]
  MoveL 836 to (440.49, 228.98, -1) mm, rotated rx -180 ry 0 rz 0 deg; joints [45.133, -53.888, 143.935, 45.128, -89.164, 0.306]
  MoveC 837 to (440.04, 228.98, -0.81) mm, rotated rx -180 ry 0 rz 0 deg; joints [45.114, -53.899, 143.915, 45.11, -89.141, 0.283] to (439.86, 228.98, -0.37) mm, rotated rx 180 ry 0 rz 0 deg; joints [45.106, -53.938, 143.912, 45.102, -89.112, 0.254]
  Set speed (500.0 mm/s)
  MoveL 838 to (439.86, 228.98, 5) mm, rotated rx 180 ry 0 rz 0 deg; joints [45.102, -54.431, 143.987, 45.103, -88.817, -0.042]
  MoveL 839 to (441.13, 293.52, 5) mm, rotated rx -180 ry 0 rz 0 deg; joints [47.658, -53.611, 140.636, 47.726, -87.128, -1.928]
  Set speed (25.4 mm/s)
  MoveL 840 to (441.13, 293.52, 1) mm, rotated rx -180 ry 0 rz 0 deg; joints [47.661, -53.265, 140.583, 47.718, -87.325, -1.712]
  MoveL 841 to (441.13, 293.52, -0.37) mm, rotated rx 180 ry 0 rz 0 deg; joints [47.662, -53.147, 140.565, 47.716, -87.392, -1.638]
  MoveC 842 to (441.13, 293.7, -0.81) mm, rotated rx -180 ry 0 rz 0 deg; joints [47.669, -53.106, 140.548, 47.722, -87.409, -1.62] to (441.13, 294.15, -1) mm, rotated rx -180 ry 0 rz 0 deg; joints [47.686, -53.083, 140.522, 47.739, -87.406, -1.624]
  Set speed (50.8 mm/s)
  MoveL 843 to (441.13, 294.79, -1) mm, rotated rx -180 ry 0 rz 0 deg; joints [47.71, -53.075, 140.487, 47.764, -87.39, -1.643]
  MoveC 844 to (441.31, 295.24, -1) mm, rotated rx -180 ry 0 rz 0 deg; joints [47.734, -53.071, 140.472, 47.788, -87.383, -1.653] to (441.76, 295.42, -1) mm, rotated rx -180 ry 0 rz 0 deg; joints [47.759, -53.075, 140.484, 47.813, -87.389, -1.647]
  MoveL 845 to (467.16, 295.42, -1) mm, rotated rx -180 ry 0 rz 0 deg; joints [48.809, -53.427, 141.731, 48.837, -88.014, -1.005]
  MoveL 846 to (467.16, 333.52, -1) mm, rotated rx 180 ry 0 rz 0 deg; joints [50.172, -52.885, 139.601, 50.253, -87.028, -2.253]
  MoveL 847 to (390.96, 333.52, -1) mm, rotated rx 180 ry 0 rz 0 deg; joints [47.137, -51.708, 135.826, 47.35, -85.135, -4.051]
  MoveL 848 to (390.96, 320.82, -1) mm, rotated rx -180 ry 0 rz 0 deg; joints [46.685, -51.912, 136.522, 46.868, -85.438, -3.659]
  MoveL 849 to (340.16, 320.82, -1) mm, rotated rx -180 ry 0 rz 0 deg; joints [44.813, -51.03, 133.833, 45.113, -84.034, -4.821]
  MoveL 850 to (340.16, 333.52, -1) mm, rotated rx 180 ry 0 rz 0 deg; joints [45.266, -50.817, 133.148, 45.603, -83.745, -5.199]
  MoveL 851 to (263.96, 333.52, -1) mm, rotated rx -180 ry 0 rz 0 deg; joints [42.67, -49.321, 128.897, 43.25, -81.492, -6.85]
  MoveL 852 to (263.96, 320.82, -1) mm, rotated rx 180 ry 0 rz 0 deg; joints [42.219, -49.545, 129.565, 42.753, -81.762, -6.485]
  MoveL 853 to (213.16, 320.82, -1) mm, rotated rx -180 ry 0 rz 0 deg; joints [40.622, -48.45, 126.566, 41.352, -80.146, -7.548]
  MoveL 854 to (213.16, 333.52, -1) mm, rotated rx 180 ry 0 rz 0 deg; joints [41.07, -48.219, 125.908, 41.853, -79.889, -7.907]
  MoveL 855 to (136.96, 333.52, -1) mm, rotated rx 180 ry 0 rz 0 deg; joints [38.849, -46.409, 121.19, 39.997, -77.345, -9.443]
  MoveL 856 to (136.96, 320.82, -1) mm, rotated rx -180 ry 0 rz 0 deg; joints [38.407, -46.648, 121.835, 39.493, -77.585, -9.086]
  MoveL 857 to (86.16, 320.82, -1) mm, rotated rx -180 ry 0 rz 0 deg; joints [37.041, -45.34, 118.522, 38.409, -75.791, -10.084]
  MoveL 858 to (86.16, 333.52, -1) mm, rotated rx -180 ry 0 rz 0 deg; joints [37.477, -45.096, 117.883, 38.914, -75.562, -10.442]
  MoveL 859 to (9.96, 333.52, -1) mm, rotated rx 180 ry 0 rz 0 deg; joints [35.57, -42.965, 112.669, 37.512, -72.76, -11.923]
  MoveL 860 to (9.96, 295.42, -1) mm, rotated rx 180 ry 0 rz 0 deg; joints [34.274, -43.705, 114.54, 35.98, -73.406, -10.849]
  MoveL 861 to (35.36, 295.42, -1) mm, rotated rx -180 ry 0 rz 0 deg; joints [34.881, -44.43, 116.319, 36.42, -74.37, -10.364]
  MoveC 862 to (48.06, 308.12, -1) mm, rotated rx -180 ry 0 rz 0 deg; joints [35.633, -44.546, 116.578, 37.164, -74.624, -10.469] to (60.76, 295.42, -1) mm, rotated rx -180 ry 0 rz 0 deg; joints [35.507, -45.133, 118.063, 36.89, -75.319, -9.878]
  MoveL 863 to (86.16, 295.42, -1) mm, rotated rx 180 ry 0 rz 0 deg; joints [36.153, -45.814, 119.774, 37.389, -76.251, -9.387]
  MoveL 864 to (162.36, 295.42, -1) mm, rotated rx -180 ry 0 rz 0 deg; joints [38.218, -47.728, 124.716, 39.065, -78.95, -7.886]
  MoveC 865 to (175.06, 308.12, -1) mm, rotated rx 180 ry 0 rz 0 deg; joints [39.038, -47.803, 124.879, 39.881, -79.134, -7.974] to (187.76, 295.42, -1) mm, rotated rx -180 ry 0 rz 0 deg; joints [38.951, -48.323, 126.301, 39.686, -79.816, -7.372]
  MoveL 866 to (289.36, 295.42, -1) mm, rotated rx -180 ry 0 rz 0 deg; joints [42.132, -50.487, 132.339, 42.501, -83.101, -5.223]
  MoveC 867 to (302.06, 308.12, -1) mm, rotated rx -180 ry 0 rz 0 deg; joints [43.026, -50.525, 132.401, 43.395, -83.204, -5.3] to (314.76, 295.42, -1) mm, rotated rx -180 ry 0 rz 0 deg; joints [42.995, -50.974, 133.774, 43.292, -83.873, -4.659]
  MoveL 868 to (416.36, 295.42, -1) mm, rotated rx 180 ry 0 rz 0 deg; joints [46.742, -52.7, 139.204, 46.83, -86.737, -2.276]
  MoveC 869 to (429.06, 308.12, -1) mm, rotated rx 180 ry 0 rz 0 deg; joints [47.712, -52.707, 139.156, 47.803, -86.743, -2.358] to (441.76, 295.42, -1) mm, rotated rx -180 ry 0 rz 0 deg; joints [47.759, -53.075, 140.484, 47.813, -87.389, -1.647]
  MoveC 870 to (441.58, 294.97, -1) mm, rotated rx -180 ry 0 rz 0 deg; joints [47.735, -53.078, 140.499, 47.789, -87.396, -1.638] to (441.13, 294.79, -1) mm, rotated rx -180 ry 0 rz 0 deg; joints [47.71, -53.075, 140.487, 47.764, -87.39, -1.643]
  MoveL 871 to (440.49, 294.79, -1) mm, rotated rx -180 ry 0 rz 0 deg; joints [47.684, -53.065, 140.455, 47.739, -87.374, -1.659]
  MoveC 872 to (440.04, 294.79, -0.81) mm, rotated rx -180 ry 0 rz 0 deg; joints [47.665, -53.075, 140.436, 47.721, -87.354, -1.681] to (439.86, 294.79, -0.37) mm, rotated rx -180 ry 0 rz 0 deg; joints [47.658, -53.111, 140.432, 47.715, -87.327, -1.709]
  Set speed (500.0 mm/s)
  MoveL 873 to (439.86, 294.79, 15) mm, rotated rx -180 ry 0 rz 0 deg; joints [47.645, -54.435, 140.629, 47.747, -86.568, -2.544]
  MoveL 874 to (439.86, 294.79, 15) mm, rotated rx -180 ry 0 rz 0 deg; joints [47.645, -54.435, 140.629, 47.747, -86.568, -2.544]
  MoveL 875 to (439.86, 294.79, 25) mm, rotated rx -180 ry 0 rz 0 deg; joints [47.637, -55.294, 140.744, 47.775, -86.067, -3.096]
